{attribute 'qualified_only'}
{attribute 'strict'}
TYPE EFeedbackMsgAttenuationELL6 :
(
	StateMsg := 1,
	PositionMsg := 10,
    IdMsg,
    CustomMsg	
);
END_TYPE

(* stored: Version 1.1.0.1, ProductVersion 3.1.4024.10
   DUT EFeedbackMsgAttenuationELL6: Id {b22775b7-898a-4144-bf86-2342dc2fb9e3} *)
